{attribute addProperty BoxType "EP7041-0002-0016"}
{attribute addProperty Id "ControlAT %Q*Control_38B054C8445.51Set_counter_valueAT %Q*UINT16217"}
{attribute addProperty CRC "2585213517"}
{attribute addProperty SizeInBites "60"}
{attribute addProperty SizeInBytes "7.5"}
TYPE ENC_Control_compact_9A173A4D :
STRUCT
	{attribute addProperty Name "Control"}
	Control AT %Q* : Control_38B054C8;
	{attribute addProperty Name "Set_counter_value"}
	Set_counter_value AT %Q* : UINT;
END_STRUCT
END_TYPE

(* stored: Version 1.2.0.0, ProductVersion 3.1.4024.9
   DUT ENC_Control_compact_9A173A4D: Id {e162d788-49db-4b6c-9ecc-651c61457c99} *)
